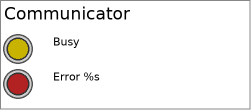
VISUALIZATION _VisuCommunicator  // 251x110
    Lamp1 (1,25 34x48), variable: ComGVL._fbTryOutCommunicator.Busy, style: Lamp-Lamp1-Yellow
    Rectangle (50,25 100x34), "Busy"
    Label (1,1 248x25), "Communicator"
    Lamp1 (1,60 34x48), variable: ComGVL._fbTryOutCommunicator.Error, style: Lamp-Lamp1-Red
    Rectangle (50,60 100x34), "Error %s", text variable: ComGVL._glErrorTable[ComGVL._fbTryOutCommunicator.ErrorID]
END_VISUALIZATION

(* stored: Version 1.1.0.1, ProductVersion 3.1.4024.2
   Visu _VisuCommunicator: Id {c4d850ec-7c66-40d5-900d-ee79eb8f6159} *)
